Universal Robots PolyScope program: SocketTCP_call_response.urp

Program interfaces_m3t1 (installation=default directory=/programs createdIn=5.11.1 lastSavedIn=5.22.0 robotSerialNumber=20205500771)
Calibrated DH parameters: a=[0.00017, -0.315777, -0.390584, 0.000089, 0.000022, 0]; d=[0.16289, -151.810109, 155.986099, -4.043122, 0.099816, 0.099706]; alpha=[1.572969, -0.001875, 0.009547, 1.571313, -1.570827, 0]; deltaTheta=[0, 0.733614, -0.631905, -0.101721, 0.000001, 0]
InitVariablesNode
BeforeStart
  'Interfaces Module 3 Task 1'
  'establish a connection, recieve a value from the server, and display it'
  conn := False
  counter := 0
  progress := False
Robot Program (runOnlyOnce=false)
  Loop While (checkContinuously=false) expression=conn≟ False
    conn := socket_open("192.168.0.5", 1701, "soc_name")
    Wait Sleep waitTime=2
    counter := counter+1
  SuppressedNode
    progress := True
  Wait Sleep waitTime=2
  str := "ready"
  Script: socket_send_string(str, "soc_name")
  Wait Sleep waitTime=2
  intake := "init"
  Loop While (checkContinuously=false) expression=(intake≟"init")  or  (intake≟"")
    intake := socket_read_string("soc_name")
    Wait Sleep waitTime=0.1
  Wait Sleep waitTime=0.5
  Popup Message (haltProgram=false inputType=Variable) variable=intake
  Wait Sleep waitTime=2
  Script: socket_close()
